FUNCTION_BLOCK RemoveMoverFromGroup EXTENDS TaskBase
VAR
	mcRemoveAxisFromGroup : MC_RemoveAxisFromGroup;
	_GroupRef : ICollisionGroup;
	_Leave: BOOL;
END_VAR

METHOD Cycle : HRESULT
VAR_INPUT
END_VAR
Cycle := S_OK;
CASE State OF
	0:
		IF _Leave THEN
			Cycle := S_PENDING;
			_Done := FALSE;
			_Error := FALSE;
			_Busy := TRUE;
			mcRemoveAxisFromGroup.Execute := TRUE;
			IF mcRemoveAxisFromGroup.Busy THEN
				State := 10;
				_Leave := FALSE;
			END_IF
		END_IF
	
	10:
		IF NOT mcRemoveAxisFromGroup.Busy THEN
			IF mcRemoveAxisFromGroup.Done THEN
				_Done := TRUE;
			ELSIF mcRemoveAxisFromGroup.Error THEN
				_Error := TRUE;
			END_IF
			_Busy := FALSE;
			mcRemoveAxisFromGroup.Execute := FALSE;
			State := 0;
			Cycle := S_OK;
		END_IF
	ELSE
		Cycle := E_FAIL;
END_CASE

mcRemoveAxisFromGroup(AxesGroup := _GroupRef.GroupRef);
END_METHOD

METHOD Execute : BOOL
VAR_INPUT
	AxisID : UDINT;
END_VAR
IF NOT _Leave THEN
	Execute := _Leave := TRUE;
	mcRemoveAxisFromGroup.IdentInGroup := UDINT_TO_IDENTINGROUP(id := AxisID);
ELSE
	Execute := false;
END_IF
END_METHOD

METHOD FB_init : BOOL
VAR_INPUT
	bInitRetains : BOOL; // if TRUE, the retain variables are initialized (warm start / cold start)
	bInCopyCode : BOOL;  // if TRUE, the instance afterwards gets moved into the copy code (online change)
	GroupRef : ICollisionGroup;
END_VAR
_GroupRef := GroupRef;
END_METHOD

END_FUNCTION_BLOCK

(* stored: Version 1.1.0.1, ProductVersion 3.1.4024.12
   POU RemoveMoverFromGroup: Id {33b40d75-d01d-4ded-8ec6-9cce1233ee05}, SpecialFunc None
   Method Cycle: Id {8ab278dc-8dad-4664-bee0-b30bd7e80670}
   Method Execute: Id {efa5d448-3299-4d10-a02c-919548e37d2d}
   Method FB_init: Id {603a2033-f770-4d8a-b85b-8ffc6acb4bdf} *)
